// TIA Portal project "tictactoe" (V16)

(* hardware
DEVICE "S7-1200 station_1"  S7-1200 Station
   slot 0: "Rack_0"  S7-1200 Rack  Rack  V1.0
   slot 1: "PLC_1"  CPU 1217C DC/DC/DC  6ES7 217-1AG40-0XB0  V4.4
DEVICE "HMI_1"  KTP900 Basic PN
   slot 0: "HMI_1"  KTP900 Basic PN  6AV2 123-2JB03-0AX0  16.0.0.0
   slot 1: "HMI_RT_1"  KTP900 Basic PN  6AV2 123-2JB03-0AX0  16.0.0.0
   slot 5: "HMI_1.IE_CP_1"  PROFINET Interface  16.0.0.0
      slot 1: "PROFINET Interface_1"  PROFINET Interface
         slot 1: "Port_1"  Port
*)

// ===== PLC "PLC_1"  CPU 1217C DC/DC/DC =====

VAR_GLOBAL   // PLC tag table "ogolne"
   "X" AT %M0.0 : Bool;
   "3x3" AT %M21.0 : Bool;
   "win" AT %M0.2 : Bool;
   "kowin" AT %M0.3 : Bool;
   "krwin" AT %M0.4 : Bool;
   "Tag_1" AT %MD0 : DWord;
   "Tag_2" AT %MD4 : DWord;
   "Tag_3" AT %MD8 : DWord;
   "Tag_4" AT %MD12 : DWord;
   "Tag_5" AT %MD15 : DWord;
   "Tag_6" AT %MW15 : Word;
   "Tag_7" AT %MW17 : Word;
   "Tag_8" AT %MB19 : Byte;
   "Tag_9" AT %MD16 : DWord;
   "reset" AT %M20.0 : Bool;
END_VAR

VAR_GLOBAL   // PLC tag table "pole 2"
   "p2" AT %M2.1 : Bool;
   "pkr2" AT %M2.2 : Bool;
   "pko2" AT %M2.3 : Bool;
END_VAR

VAR_GLOBAL   // PLC tag table "pole 3"
   "p3" AT %M3.1 : Bool;
   "pkr3" AT %M3.2 : Bool;
   "pko3" AT %M3.3 : Bool;
END_VAR

VAR_GLOBAL   // PLC tag table "pole 4"
   "p4" AT %M4.1 : Bool;
   "pkr4" AT %M4.2 : Bool;
   "pko4" AT %M4.3 : Bool;
END_VAR

VAR_GLOBAL   // PLC tag table "pole 5"
   "p5" AT %M5.1 : Bool;
   "pkr5" AT %M5.2 : Bool;
   "pko5" AT %M5.3 : Bool;
END_VAR

VAR_GLOBAL   // PLC tag table "pole 6"
   "p6" AT %M6.1 : Bool;
   "pkr6" AT %M6.2 : Bool;
   "pko6" AT %M6.3 : Bool;
END_VAR

VAR_GLOBAL   // PLC tag table "pole 7"
   "p7" AT %M7.1 : Bool;
   "pkr7" AT %M7.2 : Bool;
   "pko7" AT %M7.3 : Bool;
END_VAR

VAR_GLOBAL   // PLC tag table "pole 8"
   "p8" AT %M8.1 : Bool;
   "pkr8" AT %M8.2 : Bool;
   "pko8" AT %M8.3 : Bool;
END_VAR

VAR_GLOBAL   // PLC tag table "pole 9"
   "p9" AT %M9.1 : Bool;
   "pkr9" AT %M9.2 : Bool;
   "pko9" AT %M9.3 : Bool;
END_VAR

VAR_GLOBAL   // PLC tag table "pole 10"
   "p10" AT %M10.1 : Bool;
   "pkr10" AT %M10.2 : Bool;
   "pko10" AT %M10.3 : Bool;
END_VAR

VAR_GLOBAL   // PLC tag table "pole 11"
   "p11" AT %M11.1 : Bool;
   "pkr11" AT %M11.2 : Bool;
   "pko11" AT %M11.3 : Bool;
END_VAR

VAR_GLOBAL   // PLC tag table "pole 12"
   "p12" AT %M12.1 : Bool;
   "pkr12" AT %M12.2 : Bool;
   "pko12" AT %M12.3 : Bool;
END_VAR

VAR_GLOBAL   // PLC tag table "pole 13"
   "p13" AT %M13.1 : Bool;
   "pkr13" AT %M13.2 : Bool;
   "pko13" AT %M13.3 : Bool;
END_VAR

VAR_GLOBAL   // PLC tag table "pole 14"
   "p14" AT %M14.1 : Bool;
   "pkr14" AT %M14.2 : Bool;
   "pko14" AT %M14.3 : Bool;
END_VAR

VAR_GLOBAL   // PLC tag table "pole 15"
   "p15" AT %M15.1 : Bool;
   "pkr15" AT %M15.2 : Bool;
   "pko15" AT %M15.3 : Bool;
END_VAR

VAR_GLOBAL   // PLC tag table "pole 16"
   "p16" AT %M16.1 : Bool;
   "pkr16" AT %M16.2 : Bool;
   "pko16" AT %M16.3 : Bool;
END_VAR

VAR_GLOBAL   // PLC tag table "pole1"
   "p1" AT %M1.1 : Bool;
   "pko1" AT %M1.2 : Bool;
   "pkr1" AT %M1.3 : Bool;
END_VAR

VAR_GLOBAL   // PLC tag table "linie 4x4"
   "l1" AT %M17.1 : Bool;
   "l2" AT %M17.2 : Bool;
   "l3" AT %M17.3 : Bool;
   "l4" AT %M17.4 : Bool;
   "l5" AT %M17.5 : Bool;
   "l6" AT %M17.6 : Bool;
   "l7" AT %M17.7 : Bool;
   "l8" AT %M18.0 : Bool;
   "l9" AT %M18.1 : Bool;
   "l10" AT %M18.2 : Bool;
END_VAR

VAR_GLOBAL   // PLC tag table "linie 3x3"
   "l11" AT %M18.3 : Bool;
   "l12" AT %M18.4 : Bool;
   "l13" AT %M18.5 : Bool;
   "l14" AT %M18.6 : Bool;
   "l15" AT %M18.7 : Bool;
   "l16" AT %M19.0 : Bool;
   "l17" AT %M19.1 : Bool;
   "l18" AT %M19.2 : Bool;
END_VAR

FUNCTION "gra 4x4" : Void   // FC1, LAD
{ S7_Optimized_Access := 'TRUE' }
VERSION : 0.1
BEGIN

REGION Network 1: pole 1
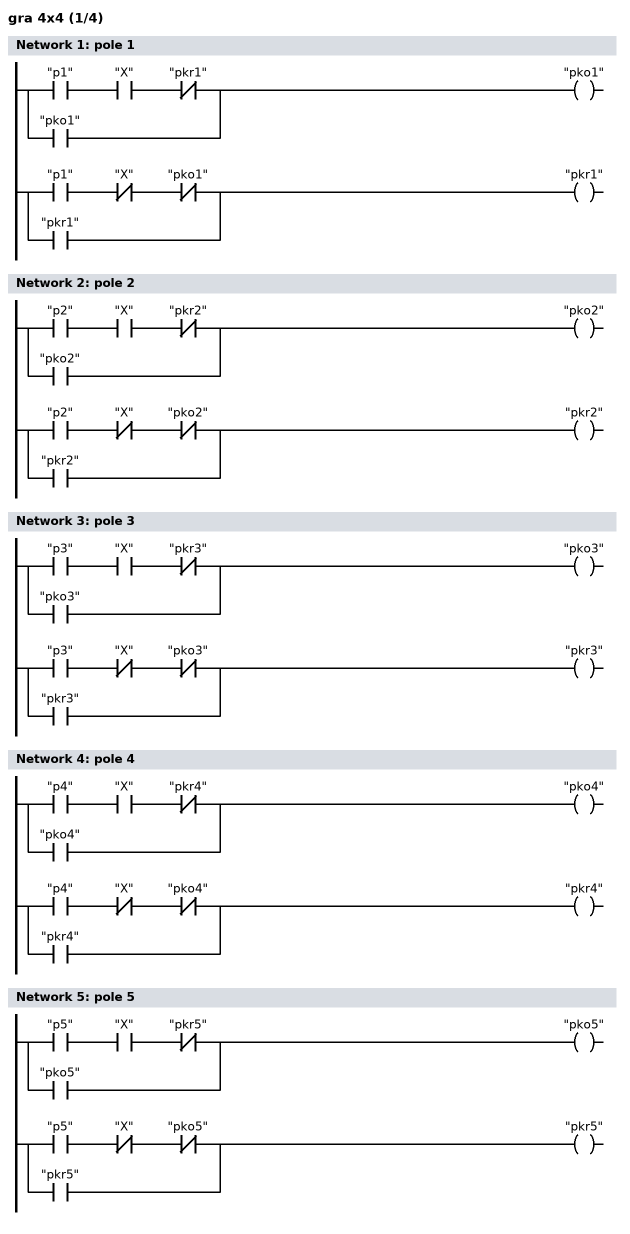
   RUNG wire#powerrail
      Contact( "p1" )
      Contact( "X" )
      I_Contact( "pkr1" )
      wire#w1
      Coil( "pko1" )
   END_RUNG
   RUNG wire#powerrail
      Contact( "pko1" )
   END_RUNG wire#w1
   RUNG wire#powerrail
      Contact( "p1" )
      I_Contact( "X" )
      I_Contact( "pko1" )
      wire#w2
      Coil( "pkr1" )
   END_RUNG
   RUNG wire#powerrail
      Contact( "pkr1" )
   END_RUNG wire#w2
   // the same network as SCL:
   "pko1" := ("p1" AND "X" AND NOT "pkr1") OR "pko1";
   "pkr1" := ("p1" AND NOT "X" AND NOT "pko1") OR "pkr1";
END_REGION

REGION Network 2: pole 2
   RUNG wire#powerrail
      Contact( "p2" )
      Contact( "X" )
      I_Contact( "pkr2" )
      wire#w1
      Coil( "pko2" )
   END_RUNG
   RUNG wire#powerrail
      Contact( "pko2" )
   END_RUNG wire#w1
   RUNG wire#powerrail
      Contact( "p2" )
      I_Contact( "X" )
      I_Contact( "pko2" )
      wire#w2
      Coil( "pkr2" )
   END_RUNG
   RUNG wire#powerrail
      Contact( "pkr2" )
   END_RUNG wire#w2
   // the same network as SCL:
   "pko2" := ("p2" AND "X" AND NOT "pkr2") OR "pko2";
   "pkr2" := ("p2" AND NOT "X" AND NOT "pko2") OR "pkr2";
END_REGION

REGION Network 3: pole 3
   RUNG wire#powerrail
      Contact( "p3" )
      Contact( "X" )
      I_Contact( "pkr3" )
      wire#w1
      Coil( "pko3" )
   END_RUNG
   RUNG wire#powerrail
      Contact( "pko3" )
   END_RUNG wire#w1
   RUNG wire#powerrail
      Contact( "p3" )
      I_Contact( "X" )
      I_Contact( "pko3" )
      wire#w2
      Coil( "pkr3" )
   END_RUNG
   RUNG wire#powerrail
      Contact( "pkr3" )
   END_RUNG wire#w2
   // the same network as SCL:
   "pko3" := ("p3" AND "X" AND NOT "pkr3") OR "pko3";
   "pkr3" := ("p3" AND NOT "X" AND NOT "pko3") OR "pkr3";
END_REGION

REGION Network 4: pole 4
   RUNG wire#powerrail
      Contact( "p4" )
      Contact( "X" )
      I_Contact( "pkr4" )
      wire#w1
      Coil( "pko4" )
   END_RUNG
   RUNG wire#powerrail
      Contact( "pko4" )
   END_RUNG wire#w1
   RUNG wire#powerrail
      Contact( "p4" )
      I_Contact( "X" )
      I_Contact( "pko4" )
      wire#w2
      Coil( "pkr4" )
   END_RUNG
   RUNG wire#powerrail
      Contact( "pkr4" )
   END_RUNG wire#w2
   // the same network as SCL:
   "pko4" := ("p4" AND "X" AND NOT "pkr4") OR "pko4";
   "pkr4" := ("p4" AND NOT "X" AND NOT "pko4") OR "pkr4";
END_REGION

REGION Network 5: pole 5
   RUNG wire#powerrail
      Contact( "p5" )
      Contact( "X" )
      I_Contact( "pkr5" )
      wire#w1
      Coil( "pko5" )
   END_RUNG
   RUNG wire#powerrail
      Contact( "pko5" )
   END_RUNG wire#w1
   RUNG wire#powerrail
      Contact( "p5" )
      I_Contact( "X" )
      I_Contact( "pko5" )
      wire#w2
      Coil( "pkr5" )
   END_RUNG
   RUNG wire#powerrail
      Contact( "pkr5" )
   END_RUNG wire#w2
   // the same network as SCL:
   "pko5" := ("p5" AND "X" AND NOT "pkr5") OR "pko5";
   "pkr5" := ("p5" AND NOT "X" AND NOT "pko5") OR "pkr5";
END_REGION

REGION Network 6: pole 6
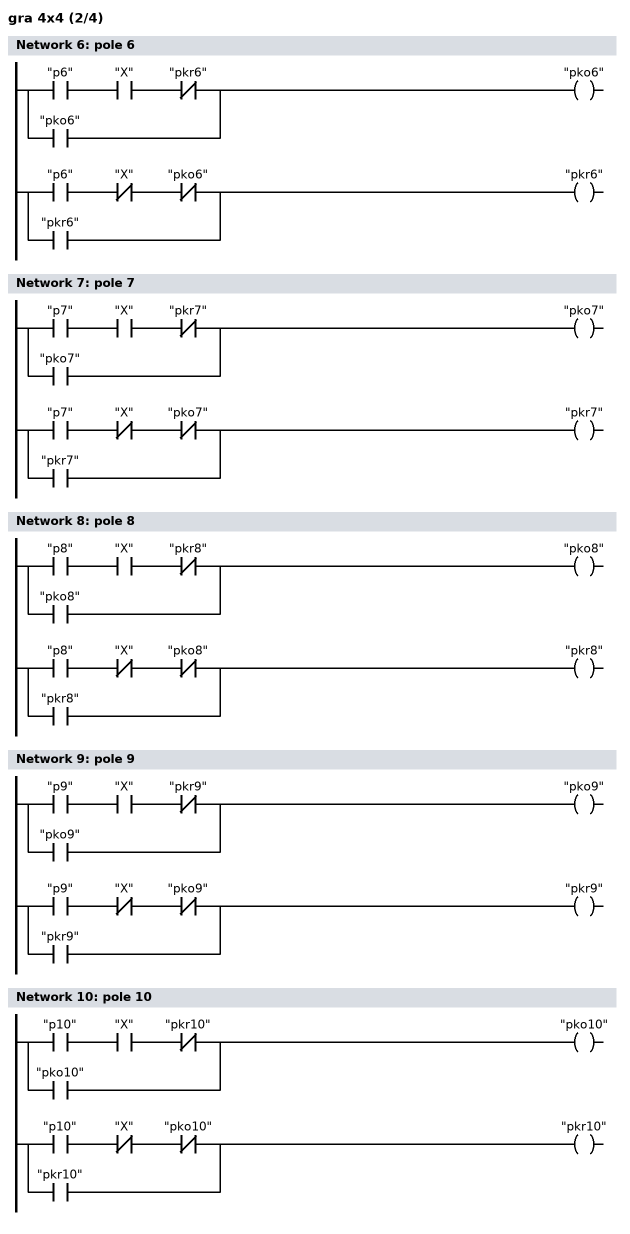
   RUNG wire#powerrail
      Contact( "p6" )
      Contact( "X" )
      I_Contact( "pkr6" )
      wire#w1
      Coil( "pko6" )
   END_RUNG
   RUNG wire#powerrail
      Contact( "pko6" )
   END_RUNG wire#w1
   RUNG wire#powerrail
      Contact( "p6" )
      I_Contact( "X" )
      I_Contact( "pko6" )
      wire#w2
      Coil( "pkr6" )
   END_RUNG
   RUNG wire#powerrail
      Contact( "pkr6" )
   END_RUNG wire#w2
   // the same network as SCL:
   "pko6" := ("p6" AND "X" AND NOT "pkr6") OR "pko6";
   "pkr6" := ("p6" AND NOT "X" AND NOT "pko6") OR "pkr6";
END_REGION

REGION Network 7: pole 7
   RUNG wire#powerrail
      Contact( "p7" )
      Contact( "X" )
      I_Contact( "pkr7" )
      wire#w1
      Coil( "pko7" )
   END_RUNG
   RUNG wire#powerrail
      Contact( "pko7" )
   END_RUNG wire#w1
   RUNG wire#powerrail
      Contact( "p7" )
      I_Contact( "X" )
      I_Contact( "pko7" )
      wire#w2
      Coil( "pkr7" )
   END_RUNG
   RUNG wire#powerrail
      Contact( "pkr7" )
   END_RUNG wire#w2
   // the same network as SCL:
   "pko7" := ("p7" AND "X" AND NOT "pkr7") OR "pko7";
   "pkr7" := ("p7" AND NOT "X" AND NOT "pko7") OR "pkr7";
END_REGION

REGION Network 8: pole 8
   RUNG wire#powerrail
      Contact( "p8" )
      Contact( "X" )
      I_Contact( "pkr8" )
      wire#w1
      Coil( "pko8" )
   END_RUNG
   RUNG wire#powerrail
      Contact( "pko8" )
   END_RUNG wire#w1
   RUNG wire#powerrail
      Contact( "p8" )
      I_Contact( "X" )
      I_Contact( "pko8" )
      wire#w2
      Coil( "pkr8" )
   END_RUNG
   RUNG wire#powerrail
      Contact( "pkr8" )
   END_RUNG wire#w2
   // the same network as SCL:
   "pko8" := ("p8" AND "X" AND NOT "pkr8") OR "pko8";
   "pkr8" := ("p8" AND NOT "X" AND NOT "pko8") OR "pkr8";
END_REGION

REGION Network 9: pole 9
   RUNG wire#powerrail
      Contact( "p9" )
      Contact( "X" )
      I_Contact( "pkr9" )
      wire#w1
      Coil( "pko9" )
   END_RUNG
   RUNG wire#powerrail
      Contact( "pko9" )
   END_RUNG wire#w1
   RUNG wire#powerrail
      Contact( "p9" )
      I_Contact( "X" )
      I_Contact( "pko9" )
      wire#w2
      Coil( "pkr9" )
   END_RUNG
   RUNG wire#powerrail
      Contact( "pkr9" )
   END_RUNG wire#w2
   // the same network as SCL:
   "pko9" := ("p9" AND "X" AND NOT "pkr9") OR "pko9";
   "pkr9" := ("p9" AND NOT "X" AND NOT "pko9") OR "pkr9";
END_REGION

REGION Network 10: pole 10
   RUNG wire#powerrail
      Contact( "p10" )
      Contact( "X" )
      I_Contact( "pkr10" )
      wire#w1
      Coil( "pko10" )
   END_RUNG
   RUNG wire#powerrail
      Contact( "pko10" )
   END_RUNG wire#w1
   RUNG wire#powerrail
      Contact( "p10" )
      I_Contact( "X" )
      I_Contact( "pko10" )
      wire#w2
      Coil( "pkr10" )
   END_RUNG
   RUNG wire#powerrail
      Contact( "pkr10" )
   END_RUNG wire#w2
   // the same network as SCL:
   "pko10" := ("p10" AND "X" AND NOT "pkr10") OR "pko10";
   "pkr10" := ("p10" AND NOT "X" AND NOT "pko10") OR "pkr10";
END_REGION

REGION Network 11: pole 11
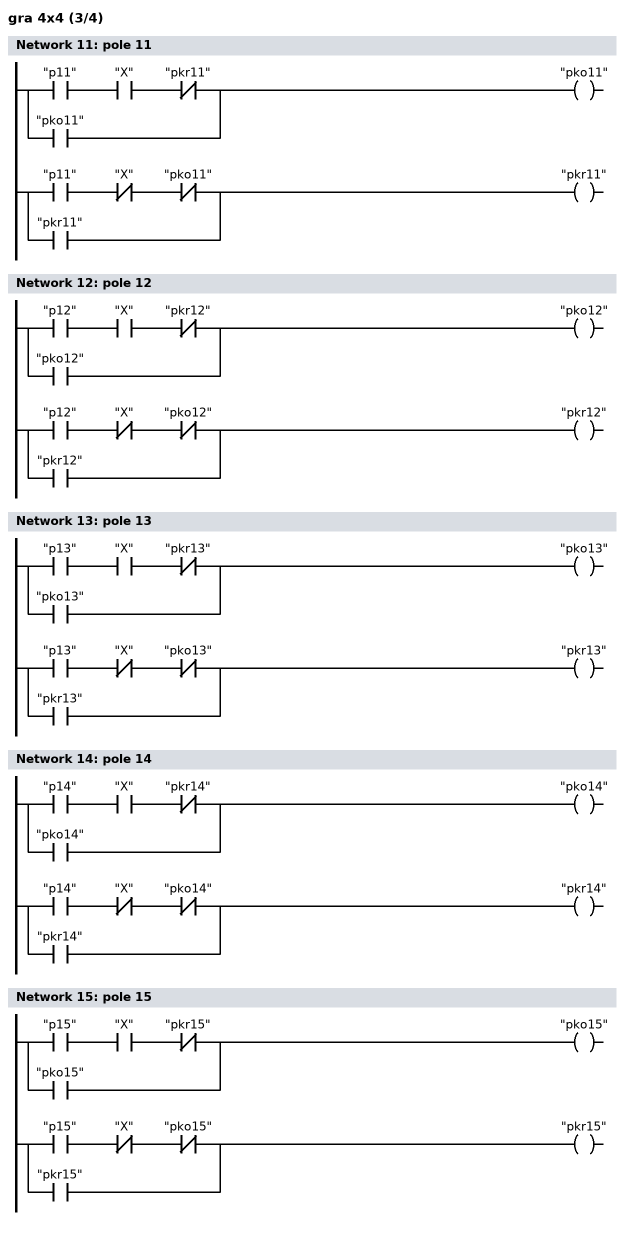
   RUNG wire#powerrail
      Contact( "p11" )
      Contact( "X" )
      I_Contact( "pkr11" )
      wire#w1
      Coil( "pko11" )
   END_RUNG
   RUNG wire#powerrail
      Contact( "pko11" )
   END_RUNG wire#w1
   RUNG wire#powerrail
      Contact( "p11" )
      I_Contact( "X" )
      I_Contact( "pko11" )
      wire#w2
      Coil( "pkr11" )
   END_RUNG
   RUNG wire#powerrail
      Contact( "pkr11" )
   END_RUNG wire#w2
   // the same network as SCL:
   "pko11" := ("p11" AND "X" AND NOT "pkr11") OR "pko11";
   "pkr11" := ("p11" AND NOT "X" AND NOT "pko11") OR "pkr11";
END_REGION

REGION Network 12: pole 12
   RUNG wire#powerrail
      Contact( "p12" )
      Contact( "X" )
      I_Contact( "pkr12" )
      wire#w1
      Coil( "pko12" )
   END_RUNG
   RUNG wire#powerrail
      Contact( "pko12" )
   END_RUNG wire#w1
   RUNG wire#powerrail
      Contact( "p12" )
      I_Contact( "X" )
      I_Contact( "pko12" )
      wire#w2
      Coil( "pkr12" )
   END_RUNG
   RUNG wire#powerrail
      Contact( "pkr12" )
   END_RUNG wire#w2
   // the same network as SCL:
   "pko12" := ("p12" AND "X" AND NOT "pkr12") OR "pko12";
   "pkr12" := ("p12" AND NOT "X" AND NOT "pko12") OR "pkr12";
END_REGION

REGION Network 13: pole 13
   RUNG wire#powerrail
      Contact( "p13" )
      Contact( "X" )
      I_Contact( "pkr13" )
      wire#w1
      Coil( "pko13" )
   END_RUNG
   RUNG wire#powerrail
      Contact( "pko13" )
   END_RUNG wire#w1
   RUNG wire#powerrail
      Contact( "p13" )
      I_Contact( "X" )
      I_Contact( "pko13" )
      wire#w2
      Coil( "pkr13" )
   END_RUNG
   RUNG wire#powerrail
      Contact( "pkr13" )
   END_RUNG wire#w2
   // the same network as SCL:
   "pko13" := ("p13" AND "X" AND NOT "pkr13") OR "pko13";
   "pkr13" := ("p13" AND NOT "X" AND NOT "pko13") OR "pkr13";
END_REGION

REGION Network 14: pole 14
   RUNG wire#powerrail
      Contact( "p14" )
      Contact( "X" )
      I_Contact( "pkr14" )
      wire#w1
      Coil( "pko14" )
   END_RUNG
   RUNG wire#powerrail
      Contact( "pko14" )
   END_RUNG wire#w1
   RUNG wire#powerrail
      Contact( "p14" )
      I_Contact( "X" )
      I_Contact( "pko14" )
      wire#w2
      Coil( "pkr14" )
   END_RUNG
   RUNG wire#powerrail
      Contact( "pkr14" )
   END_RUNG wire#w2
   // the same network as SCL:
   "pko14" := ("p14" AND "X" AND NOT "pkr14") OR "pko14";
   "pkr14" := ("p14" AND NOT "X" AND NOT "pko14") OR "pkr14";
END_REGION

REGION Network 15: pole 15
   RUNG wire#powerrail
      Contact( "p15" )
      Contact( "X" )
      I_Contact( "pkr15" )
      wire#w1
      Coil( "pko15" )
   END_RUNG
   RUNG wire#powerrail
      Contact( "pko15" )
   END_RUNG wire#w1
   RUNG wire#powerrail
      Contact( "p15" )
      I_Contact( "X" )
      I_Contact( "pko15" )
      wire#w2
      Coil( "pkr15" )
   END_RUNG
   RUNG wire#powerrail
      Contact( "pkr15" )
   END_RUNG wire#w2
   // the same network as SCL:
   "pko15" := ("p15" AND "X" AND NOT "pkr15") OR "pko15";
   "pkr15" := ("p15" AND NOT "X" AND NOT "pko15") OR "pkr15";
END_REGION

REGION Network 16: pole 16
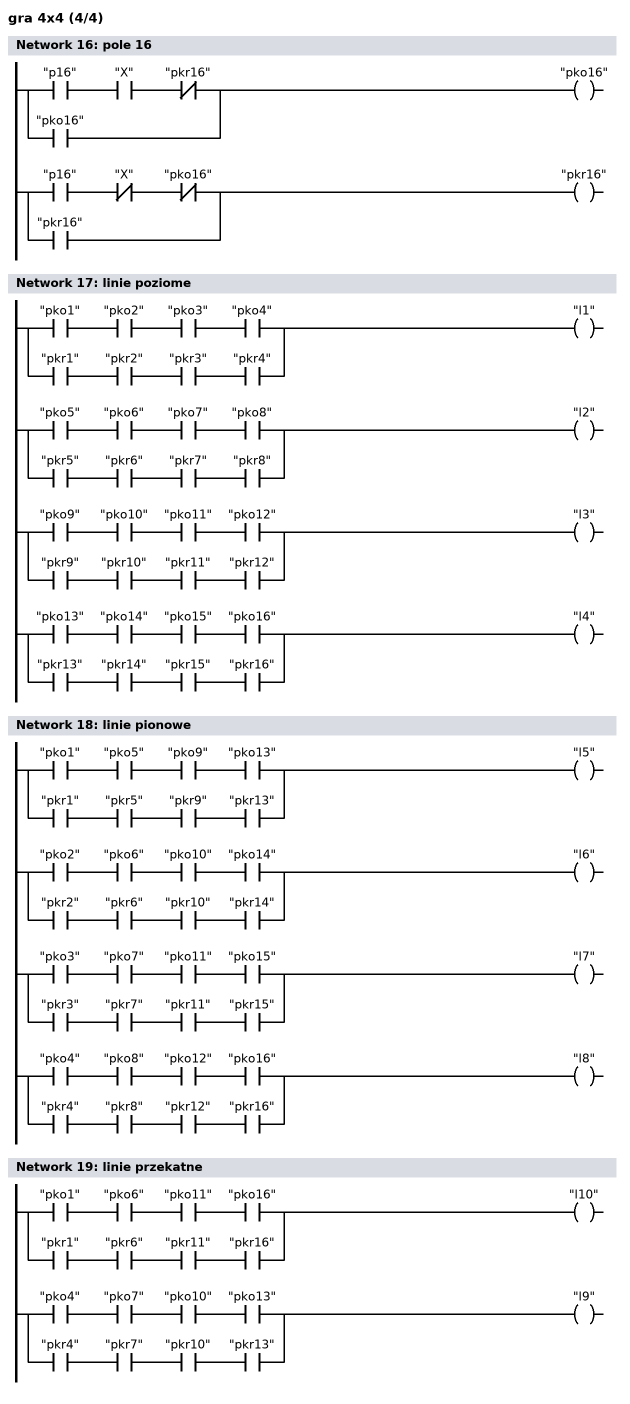
   RUNG wire#powerrail
      Contact( "p16" )
      Contact( "X" )
      I_Contact( "pkr16" )
      wire#w1
      Coil( "pko16" )
   END_RUNG
   RUNG wire#powerrail
      Contact( "pko16" )
   END_RUNG wire#w1
   RUNG wire#powerrail
      Contact( "p16" )
      I_Contact( "X" )
      I_Contact( "pko16" )
      wire#w2
      Coil( "pkr16" )
   END_RUNG
   RUNG wire#powerrail
      Contact( "pkr16" )
   END_RUNG wire#w2
   // the same network as SCL:
   "pko16" := ("p16" AND "X" AND NOT "pkr16") OR "pko16";
   "pkr16" := ("p16" AND NOT "X" AND NOT "pko16") OR "pkr16";
END_REGION

REGION Network 17: linie poziome
   RUNG wire#powerrail
      Contact( "pko1" )
      Contact( "pko2" )
      Contact( "pko3" )
      Contact( "pko4" )
      wire#w1
      Coil( "l1" )
   END_RUNG
   RUNG wire#powerrail
      Contact( "pkr1" )
      Contact( "pkr2" )
      Contact( "pkr3" )
      Contact( "pkr4" )
   END_RUNG wire#w1
   RUNG wire#powerrail
      Contact( "pko5" )
      Contact( "pko6" )
      Contact( "pko7" )
      Contact( "pko8" )
      wire#w2
      Coil( "l2" )
   END_RUNG
   RUNG wire#powerrail
      Contact( "pkr5" )
      Contact( "pkr6" )
      Contact( "pkr7" )
      Contact( "pkr8" )
   END_RUNG wire#w2
   RUNG wire#powerrail
      Contact( "pko9" )
      Contact( "pko10" )
      Contact( "pko11" )
      Contact( "pko12" )
      wire#w3
      Coil( "l3" )
   END_RUNG
   RUNG wire#powerrail
      Contact( "pkr9" )
      Contact( "pkr10" )
      Contact( "pkr11" )
      Contact( "pkr12" )
   END_RUNG wire#w3
   RUNG wire#powerrail
      Contact( "pko13" )
      Contact( "pko14" )
      Contact( "pko15" )
      Contact( "pko16" )
      wire#w4
      Coil( "l4" )
   END_RUNG
   RUNG wire#powerrail
      Contact( "pkr13" )
      Contact( "pkr14" )
      Contact( "pkr15" )
      Contact( "pkr16" )
   END_RUNG wire#w4
   // the same network as SCL:
   "l1" := ("pko1" AND "pko2" AND "pko3" AND "pko4") OR ("pkr1" AND "pkr2" AND "pkr3" AND "pkr4");
   "l2" := ("pko5" AND "pko6" AND "pko7" AND "pko8") OR ("pkr5" AND "pkr6" AND "pkr7" AND "pkr8");
   "l3" := ("pko9" AND "pko10" AND "pko11" AND "pko12") OR ("pkr9" AND "pkr10" AND "pkr11" AND "pkr12");
   "l4" := ("pko13" AND "pko14" AND "pko15" AND "pko16") OR ("pkr13" AND "pkr14" AND "pkr15" AND "pkr16");
END_REGION

REGION Network 18: linie pionowe
   RUNG wire#powerrail
      Contact( "pko1" )
      Contact( "pko5" )
      Contact( "pko9" )
      Contact( "pko13" )
      wire#w1
      Coil( "l5" )
   END_RUNG
   RUNG wire#powerrail
      Contact( "pkr1" )
      Contact( "pkr5" )
      Contact( "pkr9" )
      Contact( "pkr13" )
   END_RUNG wire#w1
   RUNG wire#powerrail
      Contact( "pko2" )
      Contact( "pko6" )
      Contact( "pko10" )
      Contact( "pko14" )
      wire#w2
      Coil( "l6" )
   END_RUNG
   RUNG wire#powerrail
      Contact( "pkr2" )
      Contact( "pkr6" )
      Contact( "pkr10" )
      Contact( "pkr14" )
   END_RUNG wire#w2
   RUNG wire#powerrail
      Contact( "pko3" )
      Contact( "pko7" )
      Contact( "pko11" )
      Contact( "pko15" )
      wire#w3
      Coil( "l7" )
   END_RUNG
   RUNG wire#powerrail
      Contact( "pkr3" )
      Contact( "pkr7" )
      Contact( "pkr11" )
      Contact( "pkr15" )
   END_RUNG wire#w3
   RUNG wire#powerrail
      Contact( "pko4" )
      Contact( "pko8" )
      Contact( "pko12" )
      Contact( "pko16" )
      wire#w4
      Coil( "l8" )
   END_RUNG
   RUNG wire#powerrail
      Contact( "pkr4" )
      Contact( "pkr8" )
      Contact( "pkr12" )
      Contact( "pkr16" )
   END_RUNG wire#w4
   // the same network as SCL:
   "l5" := ("pko1" AND "pko5" AND "pko9" AND "pko13") OR ("pkr1" AND "pkr5" AND "pkr9" AND "pkr13");
   "l6" := ("pko2" AND "pko6" AND "pko10" AND "pko14") OR ("pkr2" AND "pkr6" AND "pkr10" AND "pkr14");
   "l7" := ("pko3" AND "pko7" AND "pko11" AND "pko15") OR ("pkr3" AND "pkr7" AND "pkr11" AND "pkr15");
   "l8" := ("pko4" AND "pko8" AND "pko12" AND "pko16") OR ("pkr4" AND "pkr8" AND "pkr12" AND "pkr16");
END_REGION

REGION Network 19: linie przekatne
   RUNG wire#powerrail
      Contact( "pko1" )
      Contact( "pko6" )
      Contact( "pko11" )
      Contact( "pko16" )
      wire#w1
      Coil( "l10" )
   END_RUNG
   RUNG wire#powerrail
      Contact( "pkr1" )
      Contact( "pkr6" )
      Contact( "pkr11" )
      Contact( "pkr16" )
   END_RUNG wire#w1
   RUNG wire#powerrail
      Contact( "pko4" )
      Contact( "pko7" )
      Contact( "pko10" )
      Contact( "pko13" )
      wire#w2
      Coil( "l9" )
   END_RUNG
   RUNG wire#powerrail
      Contact( "pkr4" )
      Contact( "pkr7" )
      Contact( "pkr10" )
      Contact( "pkr13" )
   END_RUNG wire#w2
   // the same network as SCL:
   "l10" := ("pko1" AND "pko6" AND "pko11" AND "pko16") OR ("pkr1" AND "pkr6" AND "pkr11" AND "pkr16");
   "l9" := ("pko4" AND "pko7" AND "pko10" AND "pko13") OR ("pkr4" AND "pkr7" AND "pkr10" AND "pkr13");
END_REGION
END_FUNCTION

FUNCTION "gra 3x3" : Void   // FC2, LAD
{ S7_Optimized_Access := 'TRUE' }
VERSION : 0.1
BEGIN

REGION Network 1: pole 1
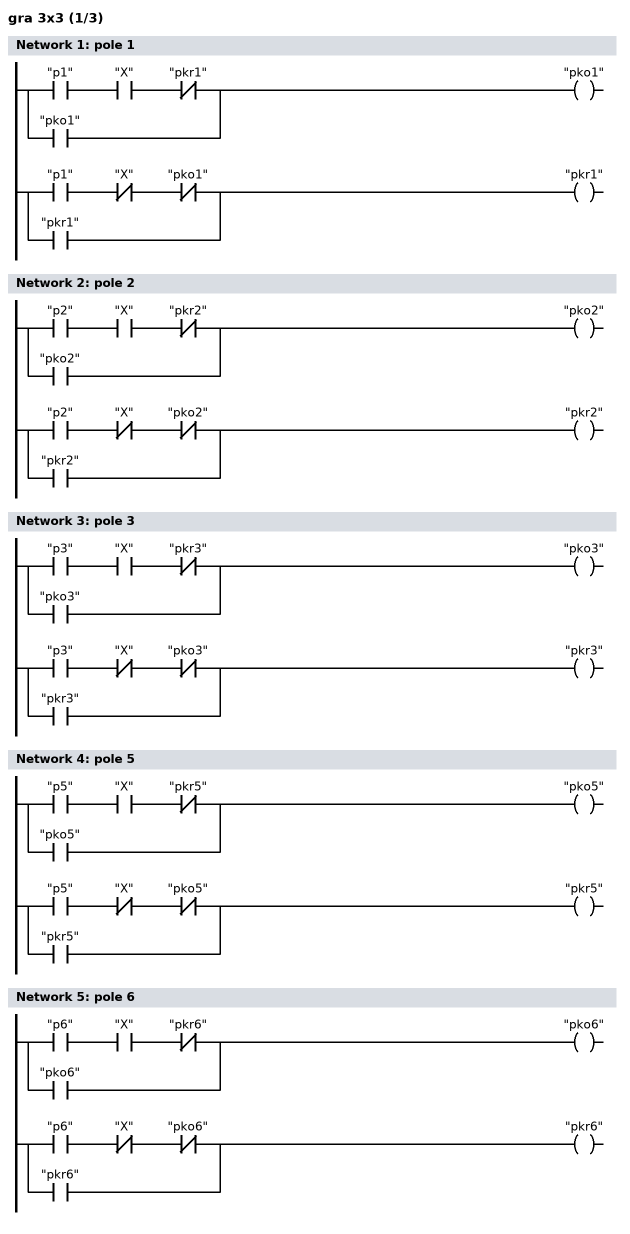
   RUNG wire#powerrail
      Contact( "p1" )
      Contact( "X" )
      I_Contact( "pkr1" )
      wire#w1
      Coil( "pko1" )
   END_RUNG
   RUNG wire#powerrail
      Contact( "pko1" )
   END_RUNG wire#w1
   RUNG wire#powerrail
      Contact( "p1" )
      I_Contact( "X" )
      I_Contact( "pko1" )
      wire#w2
      Coil( "pkr1" )
   END_RUNG
   RUNG wire#powerrail
      Contact( "pkr1" )
   END_RUNG wire#w2
   // the same network as SCL:
   "pko1" := ("p1" AND "X" AND NOT "pkr1") OR "pko1";
   "pkr1" := ("p1" AND NOT "X" AND NOT "pko1") OR "pkr1";
END_REGION

REGION Network 2: pole 2
   RUNG wire#powerrail
      Contact( "p2" )
      Contact( "X" )
      I_Contact( "pkr2" )
      wire#w1
      Coil( "pko2" )
   END_RUNG
   RUNG wire#powerrail
      Contact( "pko2" )
   END_RUNG wire#w1
   RUNG wire#powerrail
      Contact( "p2" )
      I_Contact( "X" )
      I_Contact( "pko2" )
      wire#w2
      Coil( "pkr2" )
   END_RUNG
   RUNG wire#powerrail
      Contact( "pkr2" )
   END_RUNG wire#w2
   // the same network as SCL:
   "pko2" := ("p2" AND "X" AND NOT "pkr2") OR "pko2";
   "pkr2" := ("p2" AND NOT "X" AND NOT "pko2") OR "pkr2";
END_REGION

REGION Network 3: pole 3
   RUNG wire#powerrail
      Contact( "p3" )
      Contact( "X" )
      I_Contact( "pkr3" )
      wire#w1
      Coil( "pko3" )
   END_RUNG
   RUNG wire#powerrail
      Contact( "pko3" )
   END_RUNG wire#w1
   RUNG wire#powerrail
      Contact( "p3" )
      I_Contact( "X" )
      I_Contact( "pko3" )
      wire#w2
      Coil( "pkr3" )
   END_RUNG
   RUNG wire#powerrail
      Contact( "pkr3" )
   END_RUNG wire#w2
   // the same network as SCL:
   "pko3" := ("p3" AND "X" AND NOT "pkr3") OR "pko3";
   "pkr3" := ("p3" AND NOT "X" AND NOT "pko3") OR "pkr3";
END_REGION

REGION Network 4: pole 5
   RUNG wire#powerrail
      Contact( "p5" )
      Contact( "X" )
      I_Contact( "pkr5" )
      wire#w1
      Coil( "pko5" )
   END_RUNG
   RUNG wire#powerrail
      Contact( "pko5" )
   END_RUNG wire#w1
   RUNG wire#powerrail
      Contact( "p5" )
      I_Contact( "X" )
      I_Contact( "pko5" )
      wire#w2
      Coil( "pkr5" )
   END_RUNG
   RUNG wire#powerrail
      Contact( "pkr5" )
   END_RUNG wire#w2
   // the same network as SCL:
   "pko5" := ("p5" AND "X" AND NOT "pkr5") OR "pko5";
   "pkr5" := ("p5" AND NOT "X" AND NOT "pko5") OR "pkr5";
END_REGION

REGION Network 5: pole 6
   RUNG wire#powerrail
      Contact( "p6" )
      Contact( "X" )
      I_Contact( "pkr6" )
      wire#w1
      Coil( "pko6" )
   END_RUNG
   RUNG wire#powerrail
      Contact( "pko6" )
   END_RUNG wire#w1
   RUNG wire#powerrail
      Contact( "p6" )
      I_Contact( "X" )
      I_Contact( "pko6" )
      wire#w2
      Coil( "pkr6" )
   END_RUNG
   RUNG wire#powerrail
      Contact( "pkr6" )
   END_RUNG wire#w2
   // the same network as SCL:
   "pko6" := ("p6" AND "X" AND NOT "pkr6") OR "pko6";
   "pkr6" := ("p6" AND NOT "X" AND NOT "pko6") OR "pkr6";
END_REGION

REGION Network 6: pole 7
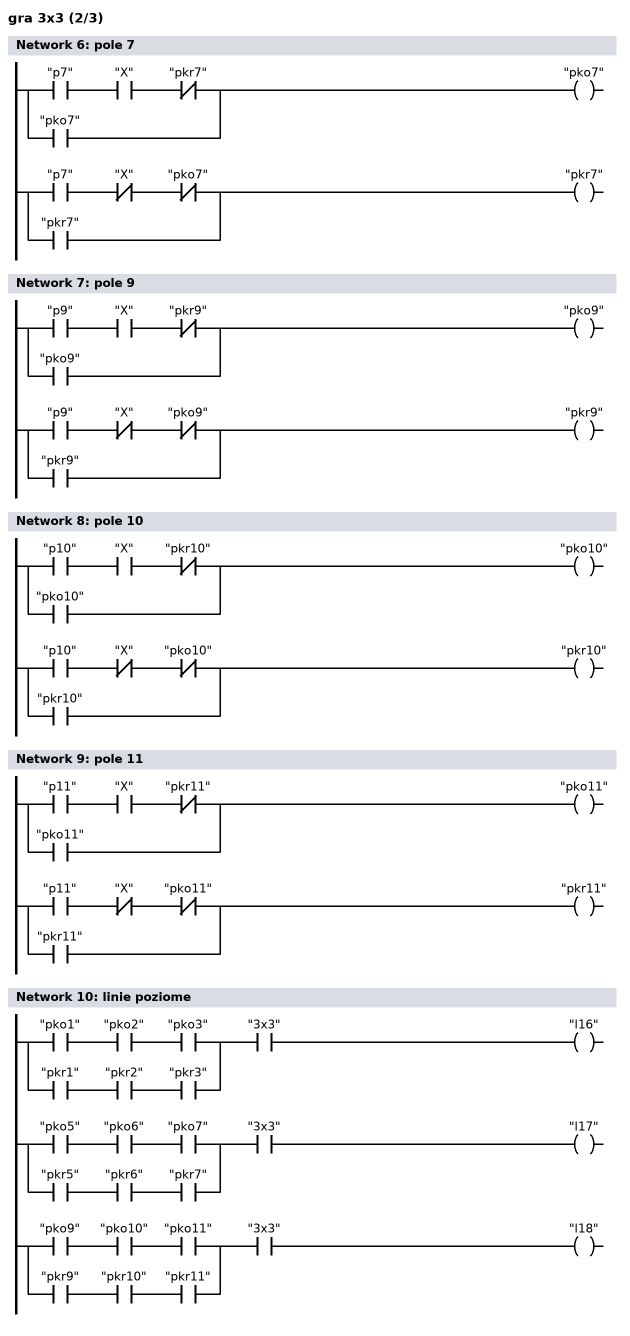
   RUNG wire#powerrail
      Contact( "p7" )
      Contact( "X" )
      I_Contact( "pkr7" )
      wire#w1
      Coil( "pko7" )
   END_RUNG
   RUNG wire#powerrail
      Contact( "pko7" )
   END_RUNG wire#w1
   RUNG wire#powerrail
      Contact( "p7" )
      I_Contact( "X" )
      I_Contact( "pko7" )
      wire#w2
      Coil( "pkr7" )
   END_RUNG
   RUNG wire#powerrail
      Contact( "pkr7" )
   END_RUNG wire#w2
   // the same network as SCL:
   "pko7" := ("p7" AND "X" AND NOT "pkr7") OR "pko7";
   "pkr7" := ("p7" AND NOT "X" AND NOT "pko7") OR "pkr7";
END_REGION

REGION Network 7: pole 9
   RUNG wire#powerrail
      Contact( "p9" )
      Contact( "X" )
      I_Contact( "pkr9" )
      wire#w1
      Coil( "pko9" )
   END_RUNG
   RUNG wire#powerrail
      Contact( "pko9" )
   END_RUNG wire#w1
   RUNG wire#powerrail
      Contact( "p9" )
      I_Contact( "X" )
      I_Contact( "pko9" )
      wire#w2
      Coil( "pkr9" )
   END_RUNG
   RUNG wire#powerrail
      Contact( "pkr9" )
   END_RUNG wire#w2
   // the same network as SCL:
   "pko9" := ("p9" AND "X" AND NOT "pkr9") OR "pko9";
   "pkr9" := ("p9" AND NOT "X" AND NOT "pko9") OR "pkr9";
END_REGION

REGION Network 8: pole 10
   RUNG wire#powerrail
      Contact( "p10" )
      Contact( "X" )
      I_Contact( "pkr10" )
      wire#w1
      Coil( "pko10" )
   END_RUNG
   RUNG wire#powerrail
      Contact( "pko10" )
   END_RUNG wire#w1
   RUNG wire#powerrail
      Contact( "p10" )
      I_Contact( "X" )
      I_Contact( "pko10" )
      wire#w2
      Coil( "pkr10" )
   END_RUNG
   RUNG wire#powerrail
      Contact( "pkr10" )
   END_RUNG wire#w2
   // the same network as SCL:
   "pko10" := ("p10" AND "X" AND NOT "pkr10") OR "pko10";
   "pkr10" := ("p10" AND NOT "X" AND NOT "pko10") OR "pkr10";
END_REGION

REGION Network 9: pole 11
   RUNG wire#powerrail
      Contact( "p11" )
      Contact( "X" )
      I_Contact( "pkr11" )
      wire#w1
      Coil( "pko11" )
   END_RUNG
   RUNG wire#powerrail
      Contact( "pko11" )
   END_RUNG wire#w1
   RUNG wire#powerrail
      Contact( "p11" )
      I_Contact( "X" )
      I_Contact( "pko11" )
      wire#w2
      Coil( "pkr11" )
   END_RUNG
   RUNG wire#powerrail
      Contact( "pkr11" )
   END_RUNG wire#w2
   // the same network as SCL:
   "pko11" := ("p11" AND "X" AND NOT "pkr11") OR "pko11";
   "pkr11" := ("p11" AND NOT "X" AND NOT "pko11") OR "pkr11";
END_REGION

REGION Network 10: linie poziome
   RUNG wire#powerrail
      Contact( "pko1" )
      Contact( "pko2" )
      Contact( "pko3" )
      wire#w1
      Contact( "3x3" )
      Coil( "l16" )
   END_RUNG
   RUNG wire#powerrail
      Contact( "pkr1" )
      Contact( "pkr2" )
      Contact( "pkr3" )
   END_RUNG wire#w1
   RUNG wire#powerrail
      Contact( "pko5" )
      Contact( "pko6" )
      Contact( "pko7" )
      wire#w2
      Contact( "3x3" )
      Coil( "l17" )
   END_RUNG
   RUNG wire#powerrail
      Contact( "pkr5" )
      Contact( "pkr6" )
      Contact( "pkr7" )
   END_RUNG wire#w2
   RUNG wire#powerrail
      Contact( "pko9" )
      Contact( "pko10" )
      Contact( "pko11" )
      wire#w3
      Contact( "3x3" )
      Coil( "l18" )
   END_RUNG
   RUNG wire#powerrail
      Contact( "pkr9" )
      Contact( "pkr10" )
      Contact( "pkr11" )
   END_RUNG wire#w3
   // the same network as SCL:
   "l16" := (("pko1" AND "pko2" AND "pko3") OR ("pkr1" AND "pkr2" AND "pkr3")) AND "3x3";
   "l17" := (("pko5" AND "pko6" AND "pko7") OR ("pkr5" AND "pkr6" AND "pkr7")) AND "3x3";
   "l18" := (("pko9" AND "pko10" AND "pko11") OR ("pkr9" AND "pkr10" AND "pkr11")) AND "3x3";
END_REGION

REGION Network 11: linie pionowe
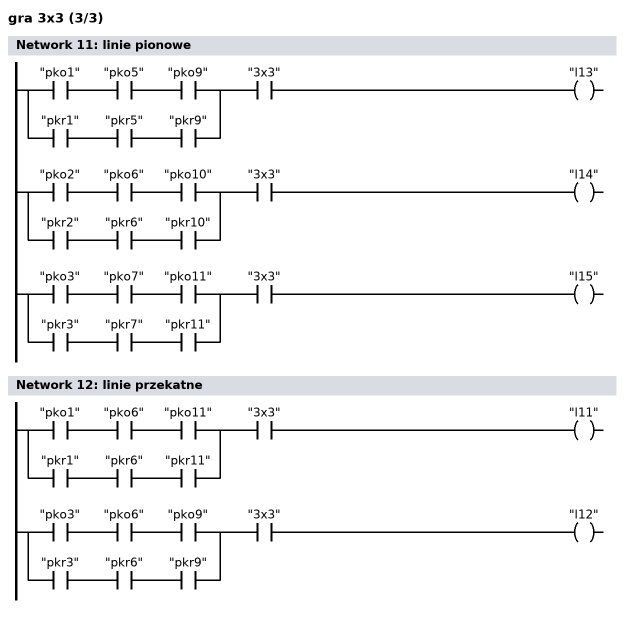
   RUNG wire#powerrail
      Contact( "pko1" )
      Contact( "pko5" )
      Contact( "pko9" )
      wire#w1
      Contact( "3x3" )
      Coil( "l13" )
   END_RUNG
   RUNG wire#powerrail
      Contact( "pkr1" )
      Contact( "pkr5" )
      Contact( "pkr9" )
   END_RUNG wire#w1
   RUNG wire#powerrail
      Contact( "pko2" )
      Contact( "pko6" )
      Contact( "pko10" )
      wire#w2
      Contact( "3x3" )
      Coil( "l14" )
   END_RUNG
   RUNG wire#powerrail
      Contact( "pkr2" )
      Contact( "pkr6" )
      Contact( "pkr10" )
   END_RUNG wire#w2
   RUNG wire#powerrail
      Contact( "pko3" )
      Contact( "pko7" )
      Contact( "pko11" )
      wire#w3
      Contact( "3x3" )
      Coil( "l15" )
   END_RUNG
   RUNG wire#powerrail
      Contact( "pkr3" )
      Contact( "pkr7" )
      Contact( "pkr11" )
   END_RUNG wire#w3
   // the same network as SCL:
   "l13" := (("pko1" AND "pko5" AND "pko9") OR ("pkr1" AND "pkr5" AND "pkr9")) AND "3x3";
   "l14" := (("pko2" AND "pko6" AND "pko10") OR ("pkr2" AND "pkr6" AND "pkr10")) AND "3x3";
   "l15" := (("pko3" AND "pko7" AND "pko11") OR ("pkr3" AND "pkr7" AND "pkr11")) AND "3x3";
END_REGION

REGION Network 12: linie przekatne
   RUNG wire#powerrail
      Contact( "pko1" )
      Contact( "pko6" )
      Contact( "pko11" )
      wire#w1
      Contact( "3x3" )
      Coil( "l11" )
   END_RUNG
   RUNG wire#powerrail
      Contact( "pkr1" )
      Contact( "pkr6" )
      Contact( "pkr11" )
   END_RUNG wire#w1
   RUNG wire#powerrail
      Contact( "pko3" )
      Contact( "pko6" )
      Contact( "pko9" )
      wire#w2
      Contact( "3x3" )
      Coil( "l12" )
   END_RUNG
   RUNG wire#powerrail
      Contact( "pkr3" )
      Contact( "pkr6" )
      Contact( "pkr9" )
   END_RUNG wire#w2
   // the same network as SCL:
   "l11" := (("pko1" AND "pko6" AND "pko11") OR ("pkr1" AND "pkr6" AND "pkr11")) AND "3x3";
   "l12" := (("pko3" AND "pko6" AND "pko9") OR ("pkr3" AND "pkr6" AND "pkr9")) AND "3x3";
END_REGION
END_FUNCTION

FUNCTION "wygrana" : Void   // FC3, LAD
{ S7_Optimized_Access := 'TRUE' }
VERSION : 0.1
BEGIN

REGION Network 1: wygranko
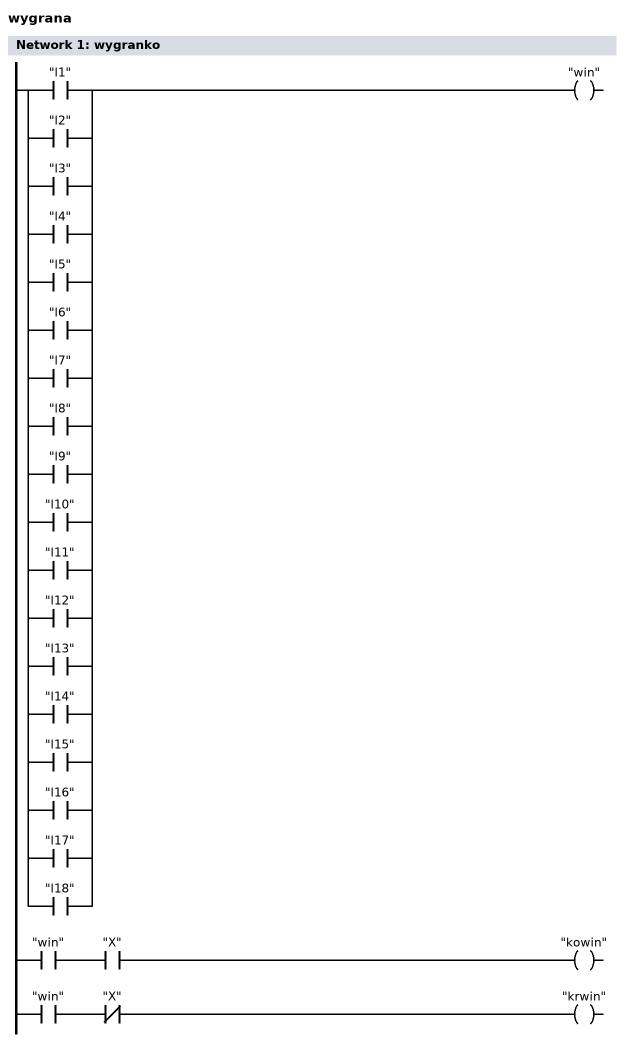
   RUNG wire#powerrail
      Contact( "l1" )
      wire#w1
      Coil( "win" )
   END_RUNG
   RUNG wire#powerrail
      Contact( "l2" )
   END_RUNG wire#w1
   RUNG wire#powerrail
      Contact( "l3" )
   END_RUNG wire#w1
   RUNG wire#powerrail
      Contact( "l4" )
   END_RUNG wire#w1
   RUNG wire#powerrail
      Contact( "l5" )
   END_RUNG wire#w1
   RUNG wire#powerrail
      Contact( "l6" )
   END_RUNG wire#w1
   RUNG wire#powerrail
      Contact( "l7" )
   END_RUNG wire#w1
   RUNG wire#powerrail
      Contact( "l8" )
   END_RUNG wire#w1
   RUNG wire#powerrail
      Contact( "l9" )
   END_RUNG wire#w1
   RUNG wire#powerrail
      Contact( "l10" )
   END_RUNG wire#w1
   RUNG wire#powerrail
      Contact( "l11" )
   END_RUNG wire#w1
   RUNG wire#powerrail
      Contact( "l12" )
   END_RUNG wire#w1
   RUNG wire#powerrail
      Contact( "l13" )
   END_RUNG wire#w1
   RUNG wire#powerrail
      Contact( "l14" )
   END_RUNG wire#w1
   RUNG wire#powerrail
      Contact( "l15" )
   END_RUNG wire#w1
   RUNG wire#powerrail
      Contact( "l16" )
   END_RUNG wire#w1
   RUNG wire#powerrail
      Contact( "l17" )
   END_RUNG wire#w1
   RUNG wire#powerrail
      Contact( "l18" )
   END_RUNG wire#w1
   RUNG wire#powerrail
      Contact( "win" )
      Contact( "X" )
      Coil( "kowin" )
   END_RUNG
   RUNG wire#powerrail
      Contact( "win" )
      I_Contact( "X" )
      Coil( "krwin" )
   END_RUNG
   // the same network as SCL:
   "win" := "l1" OR "l2" OR "l3" OR "l4" OR "l5" OR "l6" OR "l7" OR "l8" OR "l9" OR "l10" OR "l11" OR "l12" OR "l13" OR "l14" OR "l15" OR "l16" OR "l17" OR "l18";
   "kowin" := "win" AND "X";
   "krwin" := "win" AND NOT "X";
END_REGION
END_FUNCTION

FUNCTION "wyczysc_plansze" : Void   // FC4, LAD
{ S7_Optimized_Access := 'TRUE' }
VERSION : 0.1
BEGIN

REGION Network 1
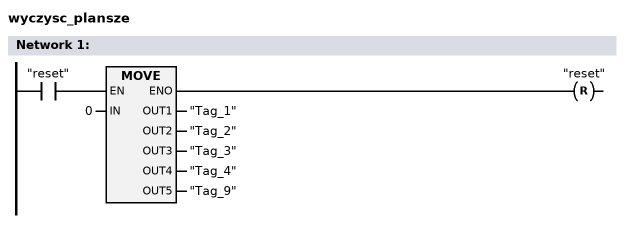
   RUNG wire#powerrail
      Contact( "reset" )
      Move(in := 0, out1 => "Tag_1", out2 => "Tag_2", out3 => "Tag_3", out4 => "Tag_4", out5 => "Tag_9")
      R_Coil( "reset" )
   END_RUNG
   // the same network as SCL:
   IF "reset" THEN
       "Tag_1" := 0;
       "Tag_2" := 0;
       "Tag_3" := 0;
       "Tag_4" := 0;
       "Tag_9" := 0;
       "reset" := FALSE;
   END_IF;
END_REGION
END_FUNCTION

ORGANIZATION_BLOCK "Main"   // OB1, LAD, ProgramCycle
TITLE = "Main Program Sweep (Cycle)"
{ S7_Optimized_Access := 'TRUE' }
VERSION : 0.1
   VAR_INPUT
      Initial_Call : Bool;   // Initial call of this OB
      Remanence : Bool;   // =True, if remanent data are available
   END_VAR
BEGIN

REGION Network 1
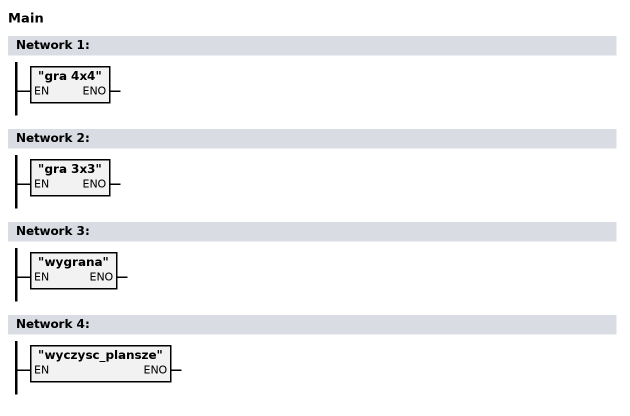
   RUNG wire#powerrail
      "gra 4x4"()
   END_RUNG
   // the same network as SCL:
   "gra 4x4"();
END_REGION

REGION Network 2
   RUNG wire#powerrail
      "gra 3x3"()
   END_RUNG
   // the same network as SCL:
   "gra 3x3"();
END_REGION

REGION Network 3
   RUNG wire#powerrail
      "wygrana"()
   END_RUNG
   // the same network as SCL:
   "wygrana"();
END_REGION

REGION Network 4
   RUNG wire#powerrail
      "wyczysc_plansze"()
   END_RUNG
   // the same network as SCL:
   "wyczysc_plansze"();
END_REGION
END_ORGANIZATION_BLOCK

(* ===== HMI "HMI_RT_1" =====
system functions are stored by id; their names below are inferred from use
connection "HMI_Connection_1": ETHERNET, SMART_S7_1200_OMS

HMI tags "Default tag table"
   "Tag_ScreenNumber" : UInt, internal
   "X" : Bool = PLC X AT %M0.0, 100 ms
   "p1" : Bool = PLC p1 AT %M1.1, 1 s
   "p2" : Bool = PLC p2 AT %M2.1, 1 s
   "pko1" : Bool = PLC pko1 AT %M1.2, 1 s
   "pkr1" : Bool = PLC pkr1 AT %M1.3, 1 s
   "pkr2" : Bool = PLC pkr2 AT %M2.2, 1 s
   "pko2" : Bool = PLC pko2 AT %M2.3, 1 s
   "3x3" : Bool = PLC 3x3 AT %M21.0, 1 s
   "p3" : Bool = PLC p3 AT %M3.1, 1 s
   "pkr3" : Bool = PLC pkr3 AT %M3.2, 1 s
   "pko3" : Bool = PLC pko3 AT %M3.3, 1 s
   "p4" : Bool = PLC p4 AT %M4.1, 1 s
   "pkr4" : Bool = PLC pkr4 AT %M4.2, 1 s
   "pko4" : Bool = PLC pko4 AT %M4.3, 1 s
   "p5" : Bool = PLC p5 AT %M5.1, 1 s
   "p6" : Bool = PLC p6 AT %M6.1, 1 s
   "p7" : Bool = PLC p7 AT %M7.1, 1 s
   "p8" : Bool = PLC p8 AT %M8.1, 1 s
   "p9" : Bool = PLC p9 AT %M9.1, 1 s
   "p10" : Bool = PLC p10 AT %M10.1, 1 s
   "p11" : Bool = PLC p11 AT %M11.1, 1 s
   "p12" : Bool = PLC p12 AT %M12.1, 1 s
   "p13" : Bool = PLC p13 AT %M13.1, 1 s
   "p14" : Bool = PLC p14 AT %M14.1, 1 s
   "p15" : Bool = PLC p15 AT %M15.1, 1 s
   "p16" : Bool = PLC p16 AT %M16.1, 1 s
   "pko5" : Bool = PLC pko5 AT %M5.3, 1 s
   "pko6" : Bool = PLC pko6 AT %M6.3, 1 s
   "pko7" : Bool = PLC pko7 AT %M7.3, 1 s
   "pko8" : Bool = PLC pko8 AT %M8.3, 1 s
   "pko9" : Bool = PLC pko9 AT %M9.3, 1 s
   "pko10" : Bool = PLC pko10 AT %M10.3, 1 s
   "pko11" : Bool = PLC pko11 AT %M11.3, 1 s
   "pko12" : Bool = PLC pko12 AT %M12.3, 1 s
   "pko13" : Bool = PLC pko13 AT %M13.3, 1 s
   "pko14" : Bool = PLC pko14 AT %M14.3, 1 s
   "pko15" : Bool = PLC pko15 AT %M15.3, 1 s
   "pko16" : Bool = PLC pko16 AT %M16.3, 1 s
   "pkr5" : Bool = PLC pkr5 AT %M5.2, 1 s
   "pkr6" : Bool = PLC pkr6 AT %M6.2, 1 s
   "pkr7" : Bool = PLC pkr7 AT %M7.2, 1 s
   "pkr8" : Bool = PLC pkr8 AT %M8.2, 1 s
   "pkr9" : Bool = PLC pkr9 AT %M9.2, 1 s
   "pkr10" : Bool = PLC pkr10 AT %M10.2, 1 s
   "pkr12" : Bool = PLC pkr12 AT %M12.2, 1 s
   "pkr13" : Bool = PLC pkr13 AT %M13.2, 1 s
   "pkr14" : Bool = PLC pkr14 AT %M14.2, 1 s
   "pkr15" : Bool = PLC pkr15 AT %M15.2, 1 s
   "pkr16" : Bool = PLC pkr16 AT %M16.2, 1 s
   "pkr11" : Bool = PLC pkr11 AT %M11.2, 1 s
   "l1" : Bool = PLC l1 AT %M17.1, 1 s
   "l2" : Bool = PLC l2 AT %M17.2, 1 s
   "l3" : Bool = PLC l3 AT %M17.3, 1 s
   "l4" : Bool = PLC l4 AT %M17.4, 1 s
   "l5" : Bool = PLC l5 AT %M17.5, 1 s
   "l6" : Bool = PLC l6 AT %M17.6, 1 s
   "l7" : Bool = PLC l7 AT %M17.7, 1 s
   "l8" : Bool = PLC l8 AT %M18.0, 1 s
   "l9" : Bool = PLC l9 AT %M18.1, 1 s
   "l10" : Bool = PLC l10 AT %M18.2, 1 s
   "kowin" : Bool = PLC kowin AT %M0.3, 1 s
   "krwin" : Bool = PLC krwin AT %M0.4, 1 s
   "win" : Bool = PLC win AT %M0.2, 1 s
   "l11" : Bool = PLC l11 AT %M18.3, 1 s
   "l12" : Bool = PLC l12 AT %M18.4, 1 s
   "l13" : Bool = PLC l13 AT %M18.5, 1 s
   "l14" : Bool = PLC l14 AT %M18.6, 1 s
   "l15" : Bool = PLC l15 AT %M18.7, 1 s
   "l16" : Bool = PLC l16 AT %M19.0, 1 s
   "l17" : Bool = PLC l17 AT %M19.1, 1 s
   "l18" : Bool = PLC l18 AT %M19.2, 1 s
   "reset" : Bool = PLC reset AT %M20.0, 1 s
   "si" : Bool = PLC si AT %M20.1, 1 s

Template "Template_1" 800x480
   Button "Exit" at 722,440 size 55x39; TextOff 'Exit'; PictureOff "ExitRuntime_KTP900_Basic_PN_TR"; PictureOn "ExitRuntime_KTP900_Basic_PN_TR"
      on Release: StopRuntime(0)
   Button "Template_Button" at 622,440 size 55x39; TextOff 'Text'
   Button "Template_Button_1" at 522,440 size 55x39; TextOff 'Text'
   Button "Template_Button_2" at 422,440 size 55x39; TextOff 'Text'
   Button "Template_Button_3" at 322,440 size 55x39; TextOff 'Text'
   Button "Template_Button_4" at 222,440 size 55x39; TextOff 'Text'
   Button "Alarms" at 122,440 size 55x39; TextOff 'Alarms'; PictureOff "AlarmDisplay_KTP900_Basic_PN_TR"; PictureOn "AlarmDisplay_KTP900_Basic_PN_TR"
      on Release: function_ef3f5d25("Alarm window_Unacknowledged", -1)
   Button "Start screen" at 22,440 size 55x39; TextOff 'Start screen'; PictureOff "NavigateHome_KTP900_Basic_PN_TR"; PictureOn "NavigateHome_KTP900_Basic_PN_TR"
      on Release: ActivateScreen("4x4", 0)
   SymbolicIOField "Symbolic_IO_Field_Screen" at 73,7 size 620x26; TextOff '0'; TextOn '1'; TextList "TextList_ScreenNames"
      ProcessValue <- "Tag_ScreenNumber"
      on Change: ActivateScreenByNumber("Tag_ScreenNumber", 0)
   DateTimeField "HmiScreenItemData" at 695,20 size 105x20
   DateTimeField "HmiScreenItemData_1" at 695,0 size 105x20
   GraphicView "Logo" at 0,0 size 71x40; Picture "Logo of HMI_1"

screen "4x4" 800x480, template "Template_1"
   on GenerateScreen: SetTag("Tag_ScreenNumber", 1)
   TextField "HmiScreenItemData" at 80,226 size 640x22; Text 'Text'
   Button "Button_1" at 600,60 size 120x60; TextOff 'Język'
   Button "Button_2" at 600,140 size 120x60; TextOff 'Plansza'
      on Click: InvertBit("3x3")
      on Change: InvertBit("3x3")
   Button "Button_20" at 600,220 size 120x60; TextOff 'Reset'
      on Change: SetBit("reset")
   Button "p1" at 200,60 size 80x80; TextOff 'Text'; TextOn 'x'
      on Click: InvertBit("X"); SetBit("p1")
   Button "p2" at 280,60 size 80x80; TextOff 'Text'
      on Click: InvertBit("X"); SetBit("p2")
   Button "p3" at 360,60 size 80x80; TextOff 'Text'
      on Click: InvertBit("X"); SetBit("p3")
   Button "p4" at 440,60 size 80x80; TextOff 'Text'
      on Click: InvertBit("X"); SetBit("p4")
      Visibility <- "3x3"
   Button "p5" at 200,140 size 80x80; TextOff 'Text'
      on Click: InvertBit("X"); SetBit("p5")
   Button "p6" at 280,140 size 80x80; TextOff 'Text'
      on Click: InvertBit("X"); SetBit("p6")
   Button "p7" at 360,140 size 80x80; TextOff 'Text'
      on Click: InvertBit("X"); SetBit("p7")
   Button "p8" at 440,140 size 80x80; TextOff 'Text'
      on Click: InvertBit("X"); SetBit("p8")
      Visibility <- "3x3"
   Button "p9" at 200,220 size 80x80; TextOff 'Text'
      on Click: InvertBit("X"); SetBit("p9")
   Button "p10" at 280,220 size 80x80; TextOff 'Text'
      on Click: InvertBit("X"); SetBit("p10")
   Button "p11" at 360,220 size 80x80; TextOff 'Text'
      on Click: InvertBit("X"); SetBit("p11")
   Button "p12" at 440,220 size 80x80; TextOff 'Text'
      on Click: InvertBit("X"); SetBit("p12")
      Visibility <- "3x3"
   Button "p13" at 200,300 size 80x80; TextOff 'Text'
      on Click: InvertBit("X"); SetBit("p13")
      Visibility <- "3x3"
   Button "p14" at 280,300 size 80x80; TextOff 'Text'
      on Click: InvertBit("X"); SetBit("p14")
      Visibility <- "3x3"
   Button "p15" at 360,300 size 80x80; TextOff 'Text'
      on Click: InvertBit("X"); SetBit("p15")
      Visibility <- "3x3"
   Button "p16" at 440,300 size 80x80; TextOff 'Text'
      on Click: InvertBit("X"); SetBit("p16")
      Visibility <- "3x3"
   TextField "kolko1" at 200,55 size 79x87; Text 'O'
      Visibility <- "pko1"
   TextField "kolko2" at 280,55 size 79x87; Text 'O'
      Visibility <- "pko2"
   TextField "kolko3" at 360,55 size 78x87; Text 'O'
      Visibility <- "pko3"
   TextField "kolko4" at 440,55 size 79x87; Text 'O'
      Visibility <- "pko4"
   TextField "kolko4_1" at 200,137 size 79x87; Text 'O'
      Visibility <- "pko5"
   TextField "kolko4_2" at 282,138 size 79x87; Text 'O'
      Visibility <- "pko6"
   TextField "kolko4_3" at 360,137 size 79x87; Text 'O'
      Visibility <- "pko7"
   TextField "kolko4_4" at 438,138 size 79x87; Text 'O'
      Visibility <- "pko8"
   TextField "kolko4_5" at 200,217 size 79x87; Text 'O'
      Visibility <- "pko9"
   TextField "kolko4_6" at 281,217 size 79x87; Text 'O'
      Visibility <- "pko10"
   TextField "kolko4_7" at 360,217 size 79x87; Text 'O'
      Visibility <- "pko11"
   TextField "kolko4_8" at 441,217 size 79x87; Text 'O'
      Visibility <- "pko12"
   TextField "kolko4_9" at 200,297 size 79x87; Text 'O'
      Visibility <- "pko13"
   TextField "kolko4_10" at 280,296 size 79x87; Text 'O'
      Visibility <- "pko14"
   TextField "kolko4_11" at 361,296 size 79x87; Text 'O'
      Visibility <- "pko15"
   TextField "kolko4_12" at 441,296 size 79x87; Text 'O'
      Visibility <- "pko16"
   TextField "krzyzyk1" at 200,55 size 77x87; Text 'X'
      Visibility <- "pkr1"
   TextField "krzyzyk2" at 280,55 size 77x87; Text 'X'
      Visibility <- "pkr2"
   TextField "krzyzyk3" at 361,55 size 77x87; Text 'X'
      Visibility <- "pkr3"
   TextField "krzyzyk4" at 443,55 size 77x87; Text 'X'
      Visibility <- "pkr4"
   TextField "krzyzyk4_1" at 202,139 size 77x87; Text 'X'
      Visibility <- "pkr5"
   TextField "krzyzyk4_2" at 282,138 size 77x87; Text 'X'
      Visibility <- "pkr6"
   TextField "krzyzyk4_3" at 361,137 size 77x87; Text 'X'
      Visibility <- "pkr7"
   TextField "krzyzyk4_4" at 442,138 size 77x87; Text 'X'
      Visibility <- "pkr8"
   TextField "krzyzyk4_5" at 201,218 size 77x87; Text 'X'
      Visibility <- "pkr9"
   TextField "krzyzyk4_6" at 282,218 size 77x87; Text 'X'
      Visibility <- "pkr10"
   TextField "krzyzyk4_7" at 362,217 size 77x87; Text 'X'
      Visibility <- "pkr11"
   TextField "krzyzyk4_8" at 441,217 size 77x87; Text 'X'
      Visibility <- "pkr12"
   TextField "krzyzyk4_9" at 201,297 size 77x87; Text 'X'
      Visibility <- "pkr13"
   TextField "krzyzyk4_10" at 281,297 size 77x87; Text 'X'
      Visibility <- "pkr14"
   TextField "krzyzyk4_11" at 362,297 size 77x87; Text 'X'
      Visibility <- "pkr15"
   TextField "krzyzyk4_12" at 441,299 size 77x87; Text 'X'
      Visibility <- "pkr16"
   Line "Line_1" at 240,90 size 0x260
      Visibility <- "l5"
   Line "Line_2" at 320,90 size 0x260
      Visibility <- "l6"
   Line "Line_3" at 400,90 size 0x260
      Visibility <- "l7"
   Line "Line_4" at 480,90 size 0x260
      Visibility <- "l8"
   Line "Line_5" at 230,100 size 260x0
      Visibility <- "l1"
   Line "Line_6" at 230,180 size 260x0
      Visibility <- "l2"
   Line "Line_7" at 230,260 size 260x0
      Visibility <- "l3"
   Line "Line_8" at 230,340 size 260x0
      Visibility <- "l4"
   Line "Line_9" at 230,90 size 260x260
      Visibility <- "l10"
   Line "Line_10" at 230,90 size 260x260
      Visibility <- "l9"
   Rectangle "Rectangle_1" at 196,59 size 324x321
      Visibility <- "kowin"
   Rectangle "Rectangle_2" at 247,142 size 243x161
      Visibility <- "kowin"
   TextField "Text field_1" at 269,173 size 196x34; Text 'Kółko wygrywa'
      Visibility <- "kowin"
   Button "Button_4" at 310,240 size 124x31; TextOff 'Ok'
      Visibility <- "kowin"
      on Change: SetBit("reset")
   Rectangle "Rectangle_3" at 196,59 size 324x321
      Visibility <- "krwin"
   Rectangle "Rectangle_4" at 247,142 size 243x161
      Visibility <- "krwin"
   TextField "Text field_2" at 258,173 size 223x34; Text 'Krzyżyk wygrywa'
      Visibility <- "krwin"
   Button "Button_5" at 310,240 size 124x31; TextOff 'Ok'
      Visibility <- "krwin"
      on Change: SetBit("reset")
   Line "Line_11" at 230,90 size 180x180
      Visibility <- "l11"
   Line "Line_12" at 230,90 size 180x180
      Visibility <- "l12"
   Line "Line_13" at 240,90 size 0x180
      Visibility <- "l13"
   Line "Line_14" at 320,90 size 0x180
      Visibility <- "l14"
   Line "Line_15" at 400,90 size 0x180
      Visibility <- "l15"
   Line "Line_16" at 230,100 size 180x0
      Visibility <- "l16"
   Line "Line_17" at 230,180 size 180x0
      Visibility <- "l17"
   Line "Line_18" at 230,260 size 180x0
      Visibility <- "l18"
*)